(* IEC 61131-3 sources: xPLCCore/codesys_code/Application/Robot_FBs/AxisGroupManager, 6 files *)

(* ---- AxisGroupManager.st ---- *)
//==============================================================================
// Main Function Block Definition
//==============================================================================
FUNCTION_BLOCK AxisGroupManager

VAR
    // --- Internal State & Events ---
    _preState : E_RobotState := E_RobotState.NULL;
    _eState : E_RobotState := E_RobotState.NULL;
    _nxtState : E_RobotState := E_RobotState.NULL;

    // --- Axis Configuration ---
    _agAxisGroup : REFERENCE TO AXIS_GROUP_REF_SM3; // Internal reference to the axis group
    _axReel      : REFERENCE TO AXIS_REF_SM3;       // Internal reference to the single (reel) axis

    // UnInited entry: the bus was at fault, so restart it (Update.st).
    xBusRestartNeeded : BOOL;

    // Error latch lives in GVL (GVL.LastErrorSource / GVL.LastErrorID) so
    // that both this FB (internal writes from Update) and external
    // supervisors (AxisGroupSM) can populate it without needing method/
    // property plumbing.

    // --- Motion Control Function Blocks ---
    fbPowerReel   : MC_Power;
    fbResetReel   : MC_Reset;
    bReelPowerReq : BOOL; // Flag to request power for the reel motor
    SMC_GroupPower_0:SM3_Robotics.SMC_GroupPower;
    GroupPower_Flag:BOOL:=FALSE;
    SMC_GroupDisable:SM3_Robotics.MC_GroupDisable;
    SMC_GroupReset:SM3_Robotics.MC_GroupReset;
    enable_fb:SM3_Robotics.MC_GroupEnable;
    homing_fb:FB_Homing;

    // State-local countdown timers (replaced the single `stateCD` shared
    // between Homing-done debounce and Ready-entry reset hold -- having
    // one variable for two unrelated purposes was a foot-gun).
    HomingDoneDebounceCD : INT; // homing_fb.bDone debounce in Homing
    ReadyResetHoldCD     : INT; // SMC_GroupReset hold scans on Ready entry

	// State-entry watchdogs. Reset on entry (IN:=FALSE in uidx=-1), driven
	// IN:=TRUE during the state's update. If .Q latches before the state
	// completes, fire EV_ERROR with source=<state>:timeout. Timeouts chosen
	// generously to tolerate normal hardware latency but still catch a
	// stuck bus / silent drive / missed Done latch.
	watchdogPowering      : Standard.TON;
	watchdogGroupEnabling : Standard.TON;
	watchdogHoming        : Standard.TON;
	WATCHDOG_POWERING_PT      : TIME := T#10S;
	WATCHDOG_GROUP_ENABLE_PT  : TIME := T#10S;
	WATCHDOG_HOMING_PT        : TIME := T#30S;

END_VAR
(* =========== IMPLEMENTATION =========== *)

// FB body is intentionally empty: nothing calls AxisGroupManagerFb() as
// a procedure. The cyclic Update(0) tick is invoked explicitly via
// `AxisGroupManagerFb.Update();` in UpdateAxisGroupState.st so the
// caller stays in control of WHERE in the scan the FSM advances
// (between TCP rx drain and motion dispatch). User events come in via
// `AxisGroupManagerFb.Transition(eEvent);` from VisuEventControl edge
// detect, DrainHostPackets GA_EV, and internal Update Trip helpers.

(* ---- FB_init.st ---- *)
//==============================================================================
// FB_init: Called once on startup to configure the FB instance.
//==============================================================================
METHOD FB_init : BOOL
VAR_INPUT
    bInitRetains : BOOL; // This parameter is required by the compiler
    bInCopyCode : BOOL;  // This parameter is required by the compiler

    // The robot's axis group
    agAxisGroup : REFERENCE TO AXIS_GROUP_REF_SM3;

    // The single (reel) axis
    axReel      : REFERENCE TO AXIS_REF_SM3;

END_VAR
VAR
    i : UINT;
END_VAR
(* =========== IMPLEMENTATION =========== *)

// Store the references
_agAxisGroup REF= agAxisGroup;
_axReel      REF= axReel;

FB_init := TRUE;

_eState:=E_RobotState.NULL;
_nxtState:=E_RobotState.UnInited;
Update(1);//exit old state
_preState:=_eState;
_eState:=_nxtState;
Update(-1);//enter new state

(* ---- Transition.st ---- *)
METHOD Transition : BOOL
VAR_INPUT
    eEvent : E_RobotEvent;
END_VAR
VAR_OUTPUT
	error:BOOL;
	new_state:E_RobotState;
END_VAR
VAR
	xForceReentry: BOOL;
END_VAR
(* =========== IMPLEMENTATION =========== *)

xForceReentry := FALSE;
new_state:=_eState;
CASE _eState OF
	E_RobotState.UnInited:
		CASE eEvent OF
			E_RobotEvent.EV_POWER_ON:
			 new_state:=E_RobotState.Powering;
		END_CASE

	E_RobotState.Powering:
		CASE eEvent OF
			E_RobotEvent.EV_OK:
			   new_state:=E_RobotState.Powered;
		END_CASE
		// EV_ERROR / EV_RESET intentionally NOT listed in the CASE above.
		// They fall through to the universal handler below:
		//   EV_ERROR -> Error  (controlled GroupStop fires; st=990 visible
		//                       to host so recovery UI engages)
		//   EV_RESET -> UnInited (universal reset, any state)
		// Pre-2026-06-23 code review: this CASE mapped EV_ERROR to
		// UnInited, so a fault during power-ramp (e.g. EtherCAT bus drop)
		// silently looked like a normal cold-down. GroupStopExecute is
		// gated on _eState=Error so the controlled stop never ran, and
		// the host's Error-state recovery path never engaged.
	E_RobotState.Powered:
		CASE eEvent OF
		E_RobotEvent.EV_GROUP_ENABLE:
			 new_state:=E_RobotState.GroupEnabling;
		END_CASE

	E_RobotState.GroupEnabling:
		CASE eEvent OF
		E_RobotEvent.EV_OK:
			 new_state:=E_RobotState.GroupEnabled;
		END_CASE

	E_RobotState.GroupEnabled:
		CASE eEvent OF
		E_RobotEvent.EV_HOME_GO:
			 new_state:=E_RobotState.Homing;
		E_RobotEvent.EV_HOME_GO_FORCE_SKIP:
			 // Skip-home is allowed only when the delta trio is virtual in
			 // the drives themselves (GVL.AxisSimMaskApplied, derived from
			 // the drives' bVirtual; bench mode SET_AXIS_SIM 0x07 --
			 // simulated arms can't physically home; the real reel axis
			 // doesn't home in this routine at all, so a real reel doesn't
			 // block it). 2026-10-04: the legacy GVL.bVirtualMotorsMode gate
			 // no longer counts -- it never touched the drives, so it could
			 // let real, unhomed axes into Ready.
			 IF (GVL.AxisSimMaskApplied AND 16#07) = 16#07 THEN
			     new_state:=E_RobotState.Ready;
			 END_IF
		END_CASE
	E_RobotState.Homing:
		CASE eEvent OF
		E_RobotEvent.EV_OK:
			 new_state:=E_RobotState.Ready;
		END_CASE

	E_RobotState.Ready:
		CASE eEvent OF
		E_RobotEvent.EV_HOME_GO:
			 new_state:=E_RobotState.Homing;
		END_CASE

	E_RobotState.Error:
		CASE eEvent OF
		E_RobotEvent.EV_RESET:
			 new_state:=E_RobotState.UnInited;
		END_CASE

END_CASE

IF(new_state=_eState)THEN//error/stop handling
	IF(eEvent=E_RobotEvent.EV_ERROR)THEN
		// Audit-fix: EV_ERROR while already in Error must re-execute the
		// entry actions (clear coord gate, re-pulse SMC_GroupDisable/Reset,
		// restamp LastErrorSource) so a stacked second fault doesn't get
		// masked by the first. Pre-fix new_state stayed Error and the
		// `IF(new_state<>_eState)` guard below skipped Update(-1).
		IF (_eState = E_RobotState.Error) THEN
			xForceReentry := TRUE;
		ELSE
			new_state:=E_RobotState.Error;
		END_IF
	ELSIF(eEvent=E_RobotEvent.EV_RESET)THEN
		// Universal reset: any state snaps back to UnInited. Lets operators
		// (and smoketests) re-run the FSM sequence without a cold boot.
		// Re-pulse entry actions even on UnInited self-loop -- otherwise an
		// operator hitting EV_RESET twice in a row to clear lingering state
		// has no effect on the second press.
		IF (_eState = E_RobotState.UnInited) THEN
			xForceReentry := TRUE;
		ELSE
			new_state:=E_RobotState.UnInited;
		END_IF
	END_IF

END_IF

IF(new_state<>_eState)THEN
  _nxtState:=new_state;
  Update(1);//exit old state
  _preState:=_eState;
  _eState:=_nxtState;
  Update(-1);//enter new state

ELSIF xForceReentry THEN
  // Same-state re-entry path. _preState/_eState unchanged; just re-run
  // exit-then-entry so the entry-side cleanup fires fresh.
  Update(1);
  Update(-1);
  GVL.SelfReentryCount := GVL.SelfReentryCount + 1;
END_IF

(* ---- TripPowerError.st ---- *)
METHOD TripPowerError : BOOL
VAR_INPUT
    psStateName : POINTER TO STRING;
END_VAR
(* =========== IMPLEMENTATION =========== *)
// Latch GVL.LastErrorSource + LastErrorID from whichever of the two
// power FBs flagged an error, then post EV_ERROR to drive the FSM
// into Error state. Used by Powering / Powered / GroupEnabled / Ready
// to dedupe the 8-line "which FB tripped + stamp + Transition" block
// that previously appeared verbatim in each.
// Caller still owns the OR-detection at the call site so the helper
// runs only when there IS an error -- no wasted CONCAT on the hot path.
IF SMC_GroupPower_0.Error THEN
    GVL.LastErrorSource := CONCAT(psStateName^, ':SMC_GroupPower');
    GVL.LastErrorID := TO_DWORD(SMC_GroupPower_0.ErrorID);
ELSE
    GVL.LastErrorSource := CONCAT(psStateName^, ':fbPowerReel');
    GVL.LastErrorID := TO_DWORD(fbPowerReel.ErrorID);
END_IF
Transition(E_RobotEvent.EV_ERROR);
TripPowerError := TRUE;

(* ---- TripTimeout.st ---- *)
METHOD TripTimeout : BOOL
VAR_INPUT
    psStateName : POINTER TO STRING;
END_VAR
(* =========== IMPLEMENTATION =========== *)
// Latch a "<state>:timeout" error source + drive EV_ERROR. Used by
// Powering / GroupEnabling / Homing when their state-entry watchdog
// TON .Q latches. ErrorID is zero (no underlying FB code) -- the
// source string distinguishes the kind of timeout.
GVL.LastErrorSource := CONCAT(psStateName^, ':timeout');
GVL.LastErrorID := 0;
Transition(E_RobotEvent.EV_ERROR);
TripTimeout := TRUE;

(* ---- Update.st ---- *)
METHOD Update : BOOL
VAR_INPUT
	//-1 enter, 0 update,1 exit current(_eState) state
	uidx:INT:=0;
END_VAR
VAR

END_VAR
(* =========== IMPLEMENTATION =========== *)

Update:=TRUE;

CASE _eState OF
    E_RobotState.UnInited:
        IF(uidx=-1)THEN // On Entry
            GVL.TestReelFrozen := FALSE;   // fault-injection hook (GVL)
            GroupPower_Flag := FALSE;
            bReelPowerReq   := FALSE; // Single Axis Power Flag

            // Was the bus at fault? Decided before the error latch is
            // cleared: only then does this entry restart the EtherCAT bus.
            xBusRestartNeeded := IoConfig_Globals.EtherCAT_Master_SoftMotion.xError
                OR (GVL.LastErrorSource = 'Supervisor:EtherCAT_Master')
                OR GVL.BusRestartOnReset;

            // Clear the error latch so a recovered run starts clean.
            GVL.LastErrorSource := '';
            GVL.LastErrorID     := 0;

            // Reset the coord-system gate: after any reset, operator must
            // re-call SetCoord0/SetCoord1 before G1 motion is accepted.
            GVL.CoordSystemConfigured := FALSE;

            // 2026-06-23 code-review fix: clear COORD1 tracking state on
            // UnInited entry too. Pre-fix, EV_RESET while a COORD1_BIND
            // was active looped FSM back through UnInited but left
            // Coord1Bound=TRUE with the previous cycle's PCS_1 transform
            // alive. The next frame=1 G1 then passed the
            // ProcessMotionPacket Coord1Bound gate against stale
            // calibration; subsequent COORD1_BIND was rejected with
            // 'rebind_requires_unbind' and the operator couldn't recover
            // without an explicit SYS COORD1_UNBIND.
            GVL.Coord1Bound       := FALSE;
            GVL.Coord1ExitPulse   := -1;
            GVL.Coord1BindEventId := 0;

            // Reset Group FBs
            SMC_GroupDisable(AxisGroup:=_agAxisGroup, Execute:=FALSE);
            SMC_GroupReset(AxisGroup:=_agAxisGroup, Execute:=FALSE);

            // Reset Single Axis FBs
            fbResetReel(Axis:= _axReel, Execute:=FALSE);

            // Restart the EtherCAT bus only when it was at fault. It used to
            // restart on every reset: each one put the DC out of sync for
            // ~3.4 s (3417 cycles, a 1190 us cycle; the "DC statistics
            // timeouts" the owner saw, machine 2026-09-29) and re-initialised
            // every slave, IO outputs included. GVL.BusRestartOnReset brings
            // the old behaviour back. Throttled: at most once per
            // BUS_RESTART_COOLDOWN_MS, so Error -> UnInited loops do not
            // hammer the master.
            IF xBusRestartNeeded AND ((GVL.LastBusRestartMs = 0) OR
               (AxisGroupSM.RuntimeMs - GVL.LastBusRestartMs >= GVL.BUS_RESTART_COOLDOWN_MS)) THEN
                IoConfig_Globals.EtherCAT_Master_SoftMotion.xRestart := TRUE;
                GVL.LastBusRestartMs := AxisGroupSM.RuntimeMs;
            END_IF
        END_IF

        IF(uidx=0)THEN // On Update
            SMC_GroupDisable(AxisGroup:=_agAxisGroup, Execute:=TRUE);
            SMC_GroupReset(AxisGroup:=_agAxisGroup, Execute:=TRUE);

            // Reset the single motor
            fbResetReel(Axis:= _axReel, Execute:=TRUE);

            IoConfig_Globals.EtherCAT_Master_SoftMotion();
            IoConfig_Globals.EtherCAT_Master_SoftMotion.xRestart:=FALSE;
        END_IF
        RETURN;

    E_RobotState.Powering:
        IF(uidx=-1)THEN
            GroupPower_Flag := FALSE;
            bReelPowerReq   := FALSE;
            watchdogPowering(IN := FALSE, PT := WATCHDOG_POWERING_PT);
        ELSIF(uidx=0)THEN
            GroupPower_Flag := TRUE;
            bReelPowerReq   := TRUE;
            watchdogPowering(IN := TRUE, PT := WATCHDOG_POWERING_PT);

            // Wait for BOTH the group and the reel motor to report powered
            IF(SMC_GroupPower_0.Status AND fbPowerReel.Status) THEN
                Transition(E_RobotEvent.EV_OK);
            ELSIF(SMC_GroupPower_0.Error OR fbPowerReel.Error) THEN
                TripPowerError(ADR('Powering'));
            ELSIF watchdogPowering.Q THEN
                TripTimeout(ADR('Powering'));
            END_IF
        END_IF

    E_RobotState.Powered:
        IF(uidx=-1)THEN
            GroupPower_Flag := TRUE;
            bReelPowerReq   := TRUE;
        ELSIF(uidx=0)THEN
            // Keep both drives alive while waiting for group enable command
            GroupPower_Flag := TRUE;
            bReelPowerReq   := TRUE;
            IF(SMC_GroupPower_0.Error OR fbPowerReel.Error) THEN
                TripPowerError(ADR('Powered'));
            END_IF
        END_IF

    E_RobotState.GroupEnabling:
        IF(uidx=-1)THEN
            enable_fb(AxisGroup:=_agAxisGroup, Execute:=FALSE);
            watchdogGroupEnabling(IN := FALSE, PT := WATCHDOG_GROUP_ENABLE_PT);
        ELSIF(uidx=0)THEN
            enable_fb(AxisGroup:=_agAxisGroup, Execute:=TRUE);
            watchdogGroupEnabling(IN := TRUE, PT := WATCHDOG_GROUP_ENABLE_PT);

            // Single motor is already enabled via MC_Power in previous state.
            // enable_fb.Error is its own source -- TripPowerError doesn't fit
            // (not a power FB); stamp inline. Watchdog uses the shared helper.
            IF(enable_fb.Done) THEN
                Transition(E_RobotEvent.EV_OK);
            ELSIF(enable_fb.Error) THEN
                GVL.LastErrorSource := 'GroupEnabling:enable_fb';
                GVL.LastErrorID := TO_DWORD(enable_fb.ErrorID);
                Transition(E_RobotEvent.EV_ERROR);
            ELSIF watchdogGroupEnabling.Q THEN
                TripTimeout(ADR('GroupEnabling'));
            END_IF
        END_IF

    E_RobotState.GroupEnabled:
        IF(uidx=-1)THEN
            GroupPower_Flag := TRUE;
            bReelPowerReq   := TRUE;
        ELSIF(uidx=0)THEN
            // Group is enabled, keep power asserted for normal operation
            GroupPower_Flag := TRUE;
            bReelPowerReq   := TRUE;
            IF(SMC_GroupPower_0.Error OR fbPowerReel.Error) THEN
                TripPowerError(ADR('GroupEnabled'));
            END_IF
        END_IF

    E_RobotState.Homing:
        IF(uidx=-1)THEN
            homing_fb(bExecute:=FALSE);
            HomingDoneDebounceCD := 100;
            watchdogHoming(IN := FALSE, PT := WATCHDOG_HOMING_PT);
        ELSIF(uidx=0)THEN
            GroupPower_Flag := TRUE;
            bReelPowerReq   := TRUE;
            homing_fb(bExecute:=TRUE);
            watchdogHoming(IN := TRUE, PT := WATCHDOG_HOMING_PT);
            IF(homing_fb.bDone) THEN
                HomingDoneDebounceCD := HomingDoneDebounceCD - 1;
                IF(HomingDoneDebounceCD = 0)THEN
                    Transition(E_RobotEvent.EV_OK);
                END_IF
            ELSIF(homing_fb.bError)THEN
                GVL.LastErrorSource := 'Homing:homing_fb';
                GVL.LastErrorID := 0;
                Transition(E_RobotEvent.EV_ERROR);
            ELSIF watchdogHoming.Q THEN
                TripTimeout(ADR('Homing'));
            ELSE
                HomingDoneDebounceCD := 100;
            END_IF
        ELSIF(uidx=1)THEN
            homing_fb(bExecute:=FALSE);
            watchdogHoming(IN := FALSE, PT := WATCHDOG_HOMING_PT);
        END_IF

    E_RobotState.Ready:
        IF(uidx=-1)THEN
            GroupPower_Flag := TRUE;
            bReelPowerReq   := TRUE;
            // Per-axis SMC_Homing (in FB_Homing) leaves the axis group in
            // ErrorStop once axes return to group control. Without a reset
            // pulse here, the very first motion packet after homing hits
            // the GroupErrorStop gate in AxisGroupSM.ProcessMotionPacket
            // and is NAKed. Hold Execute=TRUE for ReadyResetHoldCD scans
            // then drop.
            SMC_GroupReset(AxisGroup:=_agAxisGroup, Execute:=FALSE);
            ReadyResetHoldCD := 50;
        ELSIF(uidx=0)THEN
            GroupPower_Flag := TRUE;
            bReelPowerReq   := TRUE;
            IF ReadyResetHoldCD > 0 THEN
                SMC_GroupReset(AxisGroup:=_agAxisGroup, Execute:=TRUE);
                ReadyResetHoldCD := ReadyResetHoldCD - 1;
            ELSE
                SMC_GroupReset(AxisGroup:=_agAxisGroup, Execute:=FALSE);
            END_IF
            IF(SMC_GroupPower_0.Error OR fbPowerReel.Error) THEN
                TripPowerError(ADR('Ready'));
            END_IF
        END_IF

    E_RobotState.Error:
        // The reel stays powered while a tape move is under way
        // (GVL.ReelMoveInFlight): cutting it mid-move leaves the tape
        // between two cells. Its own fault or an E-stop stops it anyway;
        // the tracker then closes the move and the power drops.
        IF(uidx=-1)THEN
            GroupPower_Flag := FALSE;
            bReelPowerReq   := GVL.ReelMoveInFlight;

            // PH#6: clear the coord-system gate on Error entry too, not
            // just on UnInited. Without this, a Ready -> Error -> Ready
            // recovery (group reset by SMC, no operator EV_RESET) leaves
            // CoordSystemConfigured TRUE and lets G1 fire against stale
            // homing/coord state. UnInited entry still clears it for the
            // full reset path; this covers the in-place recovery case.
            GVL.CoordSystemConfigured := FALSE;

            SMC_GroupDisable(AxisGroup:=_agAxisGroup, Execute:=FALSE);
            SMC_GroupReset(AxisGroup:=_agAxisGroup, Execute:=FALSE);
            fbResetReel(Axis:= _axReel, Execute:=FALSE);
        END_IF

        IF(uidx=0)THEN
            // Hold power commands low every scan while in Error
            GroupPower_Flag := FALSE;
            bReelPowerReq   := GVL.ReelMoveInFlight;
            SMC_GroupDisable(AxisGroup:=_agAxisGroup, Execute:=TRUE);
            SMC_GroupReset(AxisGroup:=_agAxisGroup, Execute:=TRUE);
            fbResetReel(Axis:= _axReel, Execute:=NOT GVL.ReelMoveInFlight);
        END_IF
END_CASE

// --- CALL FUNCTION BLOCKS OUTSIDE THE CASE ---

// 1. Robot Group Power
SMC_GroupPower_0(
    AxisGroup    := _agAxisGroup,
    Enable       := TRUE,
    bRegulatorOn := GroupPower_Flag,
    bDriveStart  := GroupPower_Flag
);

// 2. Single Motor Power (Reel Pull)
fbPowerReel(
    Axis         := _axReel,
    Enable       := bReelPowerReq,
    bRegulatorOn := bReelPowerReq,
    bDriveStart  := bReelPowerReq
);

// 3. Single Motor Reset (tick every scan so Done/Busy/Error advance)
fbResetReel(Axis := _axReel);
